{attribute 'qualified_only'}
VAR_GLOBAL CONSTANT
	XtsHomePosition : LREAL := 600.0;
END_VAR

(* stored: Version 1.1.0.1, ProductVersion 3.1.4026.12
   GVL SystemConstants: Id {5fc408c7-6872-4334-8160-9577f942d020} *)
